// LS Electric XG5000 project: LoadWizardAreopag
// PLC LSPLC
// module base 0 slot 0: FEnet:XGL-EFMT(B) (Fast Ethernet Module, Electrical Master)
// module base 0 slot 1: Input Module:XGI-D24A/B (DC 24V Input, 32 Contacts)
// module base 0 slot 2: Output Module:XGQ-TR4A/B (Transistor Output, 32 Contacts (0.1A, Sink Output/Source Output))
// module base 0 slot 3: 64points reservation:XG-IN64

PROGRAM Main (task: Scan Program)

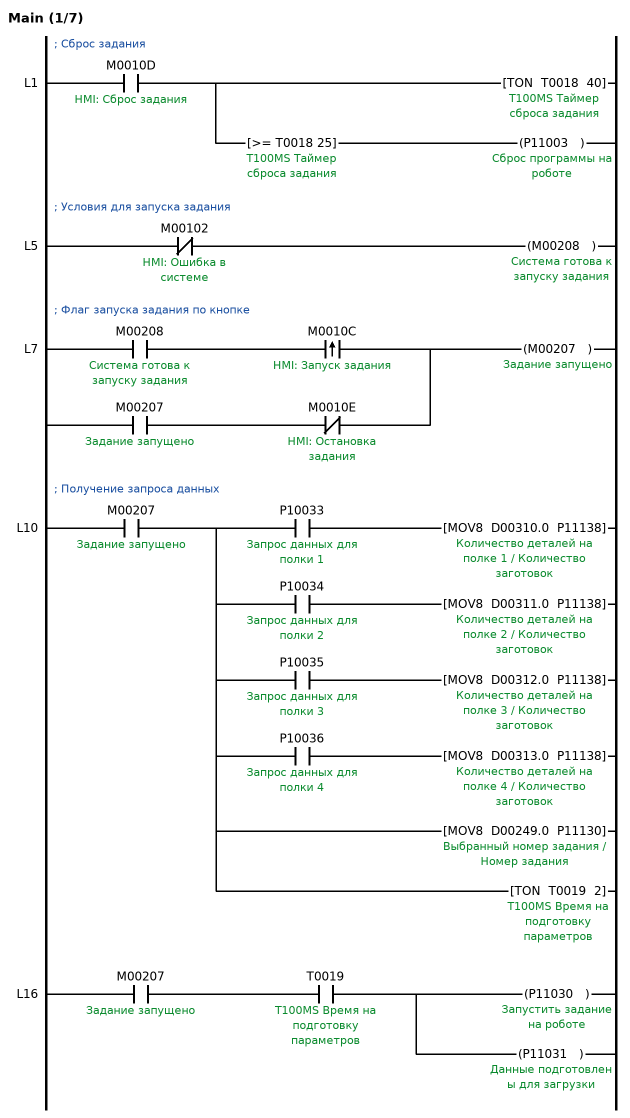
// Сброс задания
; L1
LOAD      M0010D	// HMI: Сброс задания
TON       T0018 40	// T100MS Таймер сброса задания
AND>=     T0018 25	// T100MS Таймер сброса задания
OUT       P11003	// Сброс программы на роботе
// Условия для запуска задания
; L5
LOAD NOT  M00102	// HMI: Ошибка в системе
OUT       M00208	// Система готова к запуску задания
// Флаг запуска задания по кнопке
; L7
LOAD      M00208	// Система готова к запуску задания
ANDP      M0010C	// HMI: Запуск задания
LOAD      M00207	// Задание запущено
AND NOT   M0010E	// HMI: Остановка задания
OR LOAD
OUT       M00207	// Задание запущено
// Получение запроса данных
; L10
LOAD      M00207	// Задание запущено
MPUSH
AND       P10033	// Запрос данных для полки 1
MOV8      D00310.0 P11138	// Количество деталей на полке 1 / Количество заготовок
MLOAD
AND       P10034	// Запрос данных для полки 2
MOV8      D00311.0 P11138	// Количество деталей на полке 2 / Количество заготовок
MLOAD
AND       P10035	// Запрос данных для полки 3
MOV8      D00312.0 P11138	// Количество деталей на полке 3 / Количество заготовок
MLOAD
AND       P10036	// Запрос данных для полки 4
MOV8      D00313.0 P11138	// Количество деталей на полке 4 / Количество заготовок
MPOP
MOV8      D00249.0 P11130	// Выбранный номер задания / Номер задания
TON       T0019 2	// T100MS Время на подготовку параметров
; L16
LOAD      M00207	// Задание запущено
AND       T0019	// T100MS Время на подготовку параметров
OUT       P11030	// Запустить задание на роботе
OUT       P11031	// Данные подготовлены для загрузки

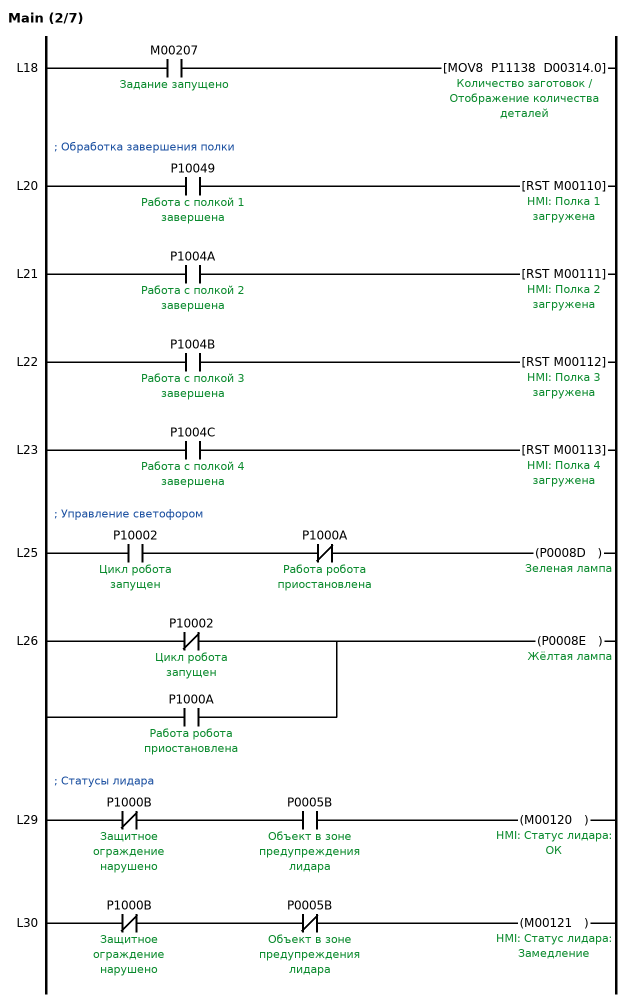
; L18
LOAD      M00207	// Задание запущено
MOV8      P11138 D00314.0	// Количество заготовок / Отображение количества деталей
// Обработка завершения полки
; L20
LOAD      P10049	// Работа с полкой 1 завершена
RST       M00110	// HMI: Полка 1 загружена
; L21
LOAD      P1004A	// Работа с полкой 2 завершена
RST       M00111	// HMI: Полка 2 загружена
; L22
LOAD      P1004B	// Работа с полкой 3 завершена
RST       M00112	// HMI: Полка 3 загружена
; L23
LOAD      P1004C	// Работа с полкой 4 завершена
RST       M00113	// HMI: Полка 4 загружена
// Управление светофором
; L25
LOAD      P10002	// Цикл робота запущен
AND NOT   P1000A	// Работа робота приостановлена
OUT       P0008D	// Зеленая лампа
; L26
LOAD NOT  P10002	// Цикл робота запущен
OR        P1000A	// Работа робота приостановлена
OUT       P0008E	// Жёлтая лампа
// Статусы лидара
; L29
LOAD NOT  P1000B	// Защитное ограждение нарушено
AND       P0005B	// Объект в зоне предупреждения лидара
OUT       M00120	// HMI: Статус лидара: ОК
; L30
LOAD NOT  P1000B	// Защитное ограждение нарушено
AND NOT   P0005B	// Объект в зоне предупреждения лидара
OUT       M00121	// HMI: Статус лидара: Замедление

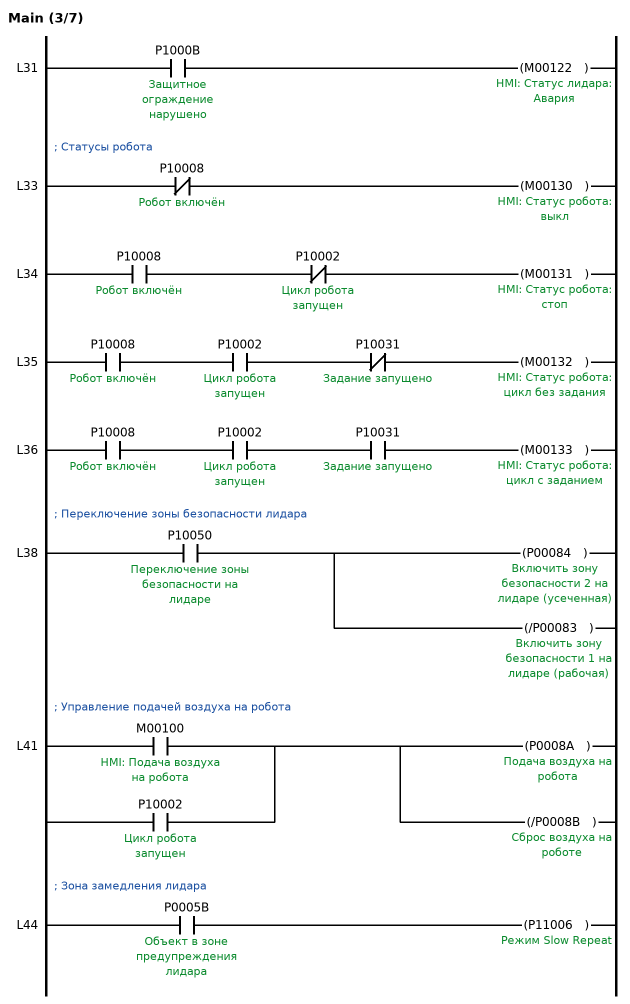
; L31
LOAD      P1000B	// Защитное ограждение нарушено
OUT       M00122	// HMI: Статус лидара: Авария
// Статусы робота
; L33
LOAD NOT  P10008	// Робот включён
OUT       M00130	// HMI: Статус робота: выкл
; L34
LOAD      P10008	// Робот включён
AND NOT   P10002	// Цикл робота запущен
OUT       M00131	// HMI: Статус робота: стоп
; L35
LOAD      P10008	// Робот включён
AND       P10002	// Цикл робота запущен
AND NOT   P10031	// Задание запущено
OUT       M00132	// HMI: Статус робота: цикл без задания
; L36
LOAD      P10008	// Робот включён
AND       P10002	// Цикл робота запущен
AND       P10031	// Задание запущено
OUT       M00133	// HMI: Статус робота: цикл с заданием
// Переключение зоны безопасности лидара 
; L38
LOAD      P10050	// Переключение зоны безопасности на лидаре
OUT       P00084	// Включить зону безопасности 2 на лидаре (усеченная)
OUT NOT   P00083	// Включить зону безопасности 1 на лидаре (рабочая)
// Управление подачей воздуха на робота
; L41
LOAD      M00100	// HMI: Подача воздуха на робота
OR        P10002	// Цикл робота запущен
OUT       P0008A	// Подача воздуха на робота
OUT NOT   P0008B	// Сброс воздуха на роботе
// Зона замедления лидара
; L44
LOAD      P0005B	// Объект в зоне предупреждения лидара
OUT       P11006	// Режим Slow Repeat

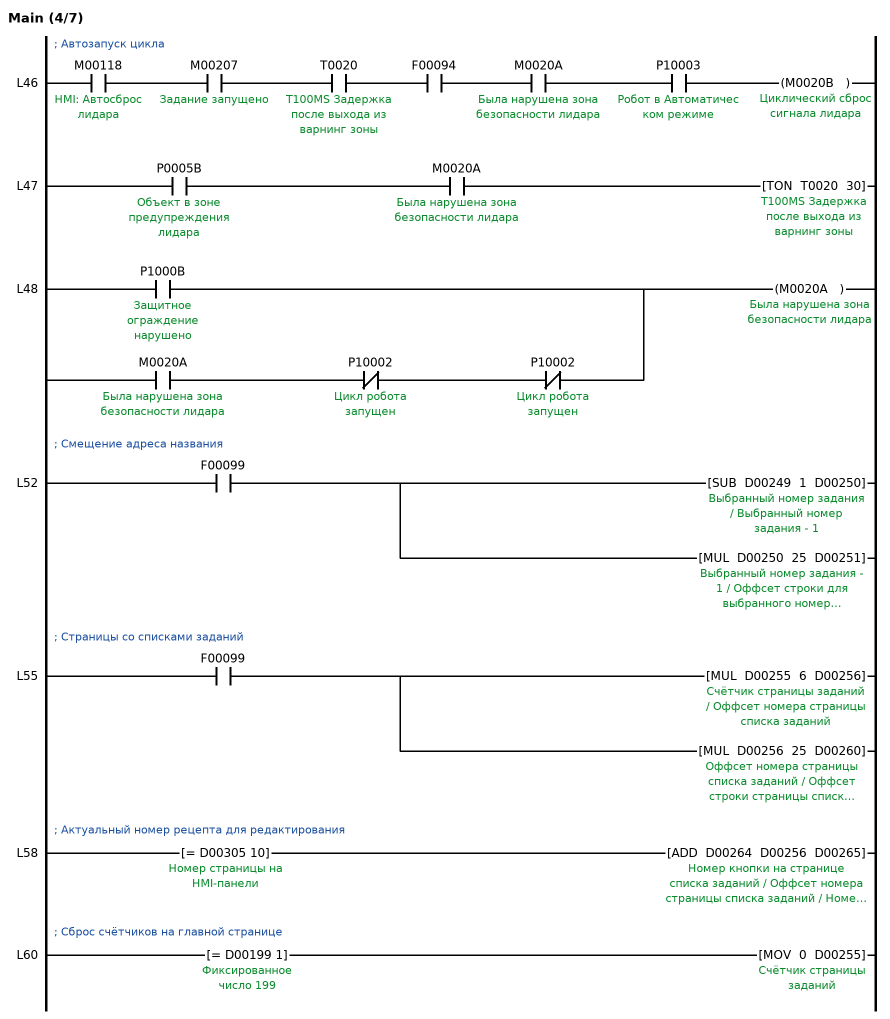
// Автозапуск цикла
; L46
LOAD      M00118	// HMI: Автосброс лидара
AND       M00207	// Задание запущено
AND       T0020	// T100MS Задержка после выхода из варнинг зоны
AND       F00094
AND       M0020A	// Была нарушена зона безопасности лидара
AND       P10003	// Робот в Автоматическом режиме
OUT       M0020B	// Циклический сброс сигнала лидара
; L47
LOAD      P0005B	// Объект в зоне предупреждения лидара
AND       M0020A	// Была нарушена зона безопасности лидара
TON       T0020 30	// T100MS Задержка после выхода из варнинг зоны
; L48
LOAD      P1000B	// Защитное ограждение нарушено
LOAD      M0020A	// Была нарушена зона безопасности лидара
AND NOT   P10002	// Цикл робота запущен
AND NOT   P10002	// Цикл робота запущен
OR LOAD
OUT       M0020A	// Была нарушена зона безопасности лидара
// Смещение адреса названия
; L52
LOAD      F00099
SUB       D00249 1 D00250	// Выбранный номер задания / Выбранный номер задания - 1
MUL       D00250 25 D00251	// Выбранный номер задания - 1 / Оффсет строки для выбранного номера названия
// Страницы со списками заданий
; L55
LOAD      F00099
MUL       D00255 6 D00256	// Счётчик страницы заданий / Оффсет номера страницы списка заданий
MUL       D00256 25 D00260	// Оффсет номера страницы списка заданий / Оффсет строки страницы списка заданий
// Актуальный номер рецепта для редактирования
; L58
LOAD=     D00305 10	// Номер страницы на HMI-панели
ADD       D00264 D00256 D00265	// Номер кнопки на странице списка заданий / Оффсет номера страницы списка заданий / Номер редактируемого задания
// Сброс счётчиков на главной странице
; L60
LOAD=     D00199 1	// Фиксированное число 199
MOV       0 D00255	// Счётчик страницы заданий

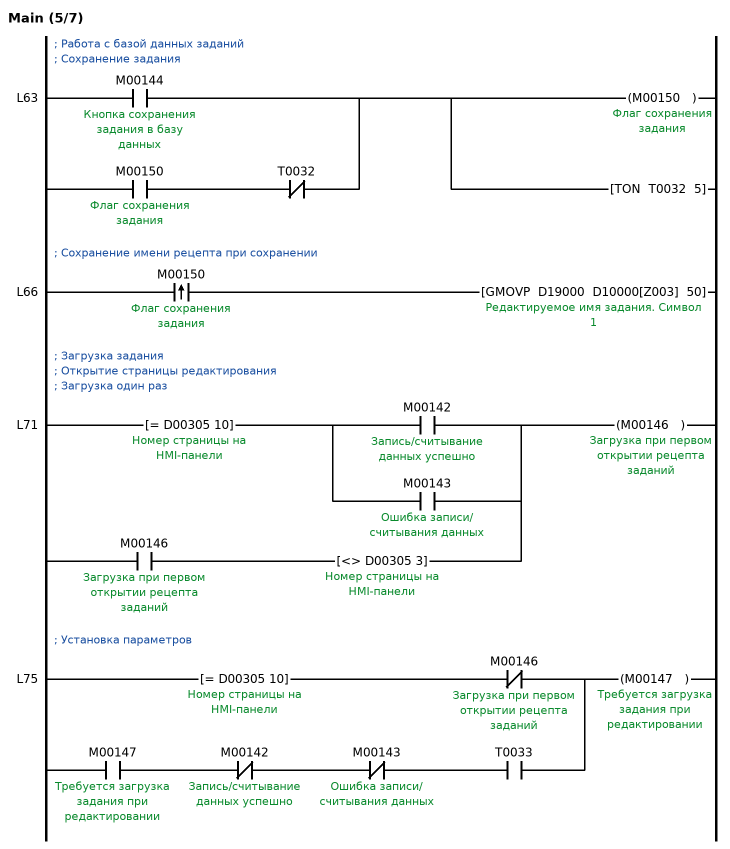
// Работа с базой данных заданий
// Сохранение задания
; L63
LOAD      M00144	// Кнопка сохранения задания в базу данных
LOAD      M00150	// Флаг сохранения задания
AND NOT   T0032
OR LOAD
OUT       M00150	// Флаг сохранения задания
TON       T0032 5
// Сохранение имени рецепта при сохранении
; L66
LOADP     M00150	// Флаг сохранения задания
GMOVP     D19000 D10000[Z003] 50	// Редактируемое имя задания. Символ 1
// Загрузка задания
// Открытие страницы редактирования
// Загрузка один раз
; L71
LOAD=     D00305 10	// Номер страницы на HMI-панели
LOAD      M00142	// Запись/считывание данных успешно
OR        M00143	// Ошибка записи/считывания данных
AND LOAD
LOAD      M00146	// Загрузка при первом открытии рецепта заданий
AND<>     D00305 3	// Номер страницы на HMI-панели
OR LOAD
OUT       M00146	// Загрузка при первом открытии рецепта заданий
// Установка параметров
; L75
LOAD=     D00305 10	// Номер страницы на HMI-панели
AND NOT   M00146	// Загрузка при первом открытии рецепта заданий
LOAD      M00147	// Требуется загрузка задания при редактировании
AND NOT   M00142	// Запись/считывание данных успешно
AND NOT   M00143	// Ошибка записи/считывания данных
AND       T0033
OR LOAD
OUT       M00147	// Требуется загрузка задания при редактировании

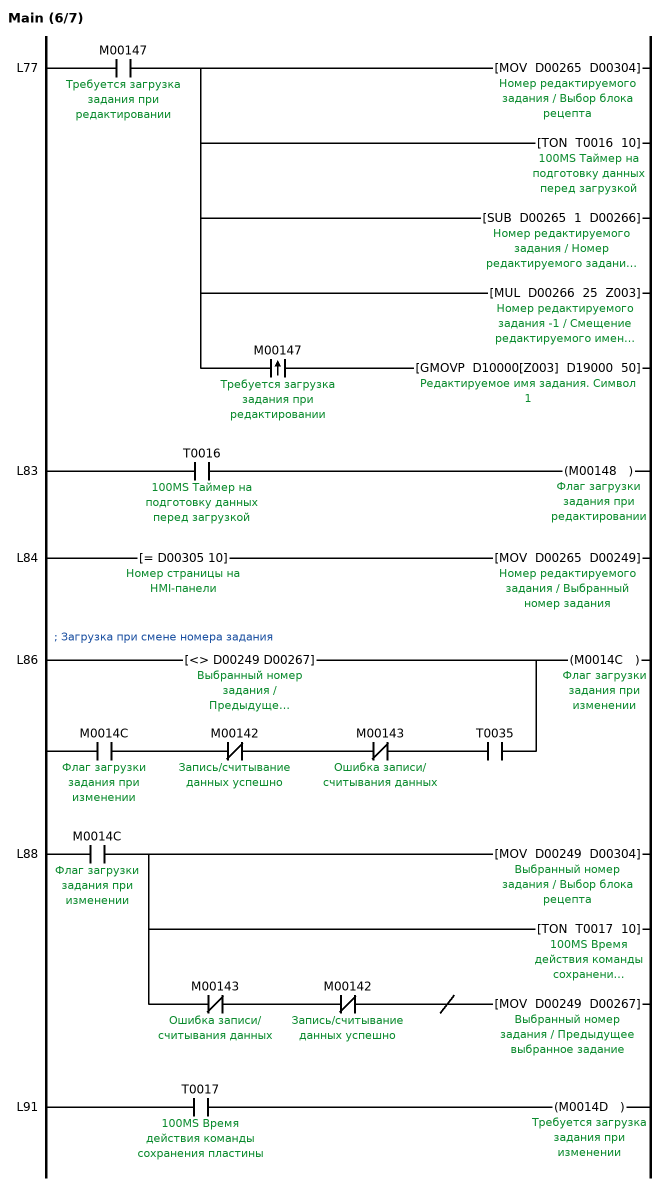
; L77
LOAD      M00147	// Требуется загрузка задания при редактировании
MOV       D00265 D00304	// Номер редактируемого задания / Выбор блока рецепта
TON       T0016 10	// 100MS Таймер на подготовку данных перед загрузкой
SUB       D00265 1 D00266	// Номер редактируемого задания / Номер редактируемого задания -1
MUL       D00266 25 Z003	// Номер редактируемого задания -1 / Смещение редактируемого имени задания
ANDP      M00147	// Требуется загрузка задания при редактировании
GMOVP     D10000[Z003] D19000 50	// Редактируемое имя задания. Символ 1
; L83
LOAD      T0016	// 100MS Таймер на подготовку данных перед загрузкой
OUT       M00148	// Флаг загрузки задания при редактировании
; L84
LOAD=     D00305 10	// Номер страницы на HMI-панели
MOV       D00265 D00249	// Номер редактируемого задания / Выбранный номер задания
// Загрузка при смене номера задания
; L86
LOAD<>    D00249 D00267	// Выбранный номер задания / Предыдущее выбранное задание
LOAD      M0014C	// Флаг загрузки задания при изменении
AND NOT   M00142	// Запись/считывание данных успешно
AND NOT   M00143	// Ошибка записи/считывания данных
AND       T0035
OR LOAD
OUT       M0014C	// Флаг загрузки задания при изменении
; L88
LOAD      M0014C	// Флаг загрузки задания при изменении
MOV       D00249 D00304	// Выбранный номер задания / Выбор блока рецепта
TON       T0017 10	// 100MS Время действия команды сохранения пластины
AND NOT   M00143	// Ошибка записи/считывания данных
AND NOT   M00142	// Запись/считывание данных успешно
NOT
MOV       D00249 D00267	// Выбранный номер задания / Предыдущее выбранное задание
; L91
LOAD      T0017	// 100MS Время действия команды сохранения пластины
OUT       M0014D	// Требуется загрузка задания при изменении

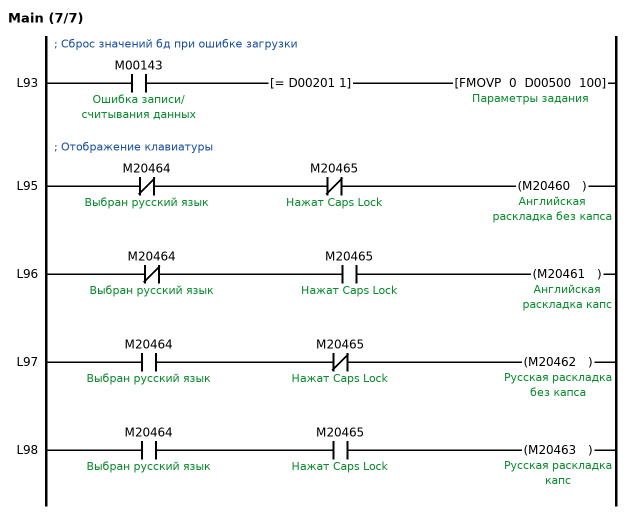
// Сброс значений бд при ошибке загрузки
; L93
LOAD      M00143	// Ошибка записи/считывания данных
AND=      D00201 1
FMOVP     0 D00500 100	// Параметры задания
// Отображение клавиатуры
; L95
LOAD NOT  M20464	// Выбран русский язык
AND NOT   M20465	// Нажат Caps Lock
OUT       M20460	// Английская раскладка без капса
; L96
LOAD NOT  M20464	// Выбран русский язык
AND       M20465	// Нажат Caps Lock
OUT       M20461	// Английская раскладка капс
; L97
LOAD      M20464	// Выбран русский язык
AND NOT   M20465	// Нажат Caps Lock
OUT       M20462	// Русская раскладка без капса
; L98
LOAD      M20464	// Выбран русский язык
AND       M20465	// Нажат Caps Lock
OUT       M20463	// Русская раскладка капс

PROGRAM CNC (task: Scan Program)

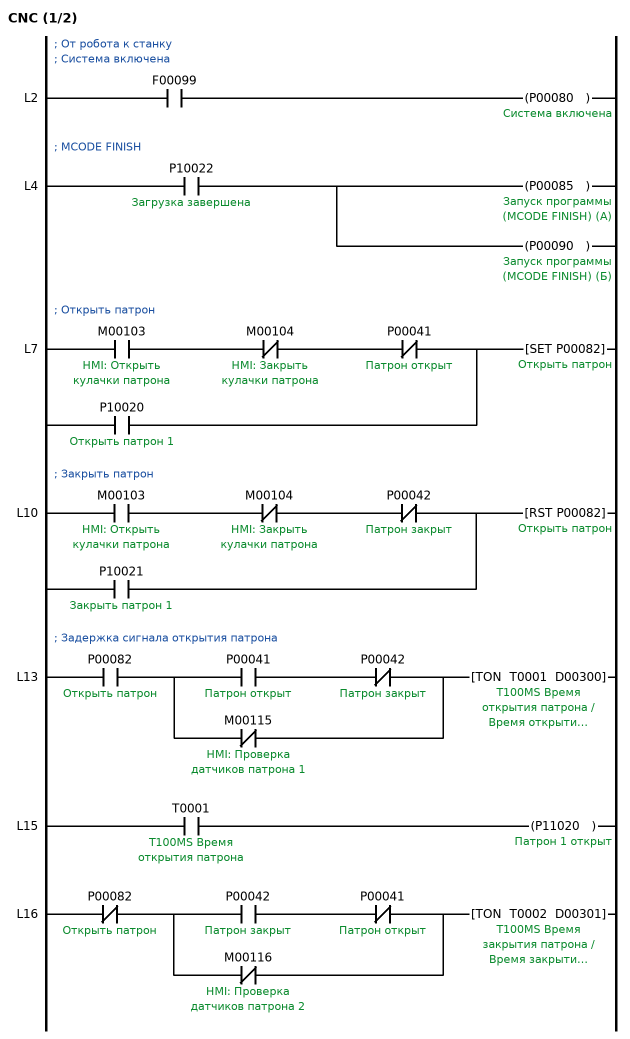
// От робота к станку
// Система включена
; L2
LOAD      F00099
OUT       P00080	// Система включена
// MCODE FINISH
; L4
LOAD      P10022	// Загрузка завершена
OUT       P00085	// Запуск программы (MCODE FINISH) (А)
OUT       P00090	// Запуск программы (MCODE FINISH) (Б)
// Открыть патрон
; L7
LOAD      M00103	// HMI: Открыть кулачки патрона
AND NOT   M00104	// HMI: Закрыть кулачки патрона
AND NOT   P00041	// Патрон открыт
OR        P10020	// Открыть патрон 1
SET       P00082	// Открыть патрон
// Закрыть патрон
; L10
LOAD      M00103	// HMI: Открыть кулачки патрона
AND NOT   M00104	// HMI: Закрыть кулачки патрона
AND NOT   P00042	// Патрон закрыт
OR        P10021	// Закрыть патрон 1
RST       P00082	// Открыть патрон
// Задержка сигнала открытия патрона
; L13
LOAD      P00082	// Открыть патрон
LOAD      P00041	// Патрон открыт
AND NOT   P00042	// Патрон закрыт
OR NOT    M00115	// HMI: Проверка датчиков патрона 1
AND LOAD
TON       T0001 D00300	// T100MS Время открытия патрона / Время открытия патрона (сек)
; L15
LOAD      T0001	// T100MS Время открытия патрона
OUT       P11020	// Патрон 1 открыт
; L16
LOAD NOT  P00082	// Открыть патрон
LOAD      P00042	// Патрон закрыт
AND NOT   P00041	// Патрон открыт
OR NOT    M00116	// HMI: Проверка датчиков патрона 2
AND LOAD
TON       T0002 D00301	// T100MS Время закрытия патрона / Время закрытия патрона (сек)

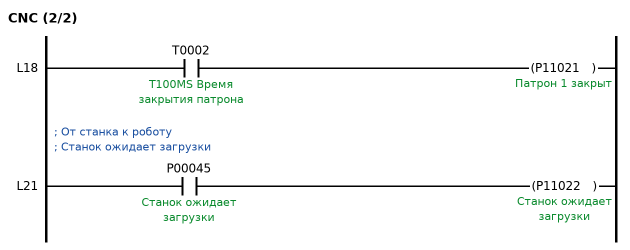
; L18
LOAD      T0002	// T100MS Время закрытия патрона
OUT       P11021	// Патрон 1 закрыт
// От станка к роботу
// Станок ожидает загрузки
; L21
LOAD      P00045	// Станок ожидает загрузки
OUT       P11022	// Станок ожидает загрузки

PROGRAM Error (task: Scan Program)

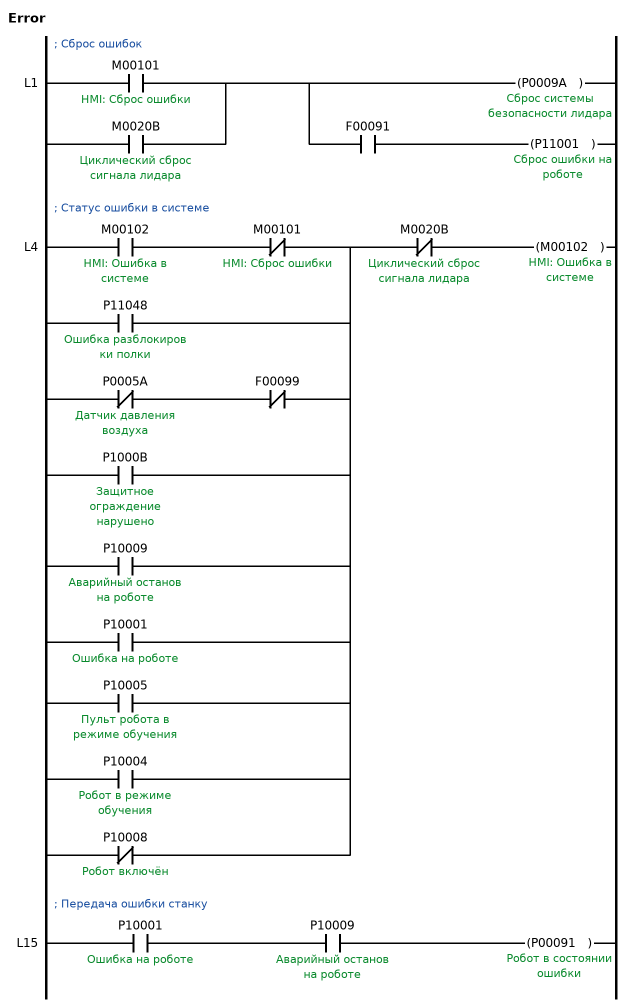
// Сброс ошибок
; L1
LOAD      M00101	// HMI: Сброс ошибки
OR        M0020B	// Циклический сброс сигнала лидара
OUT       P0009A	// Сброс системы безопасности лидара
AND       F00091
OUT       P11001	// Сброс ошибки на роботе
// Статус ошибки в системе
; L4
LOAD      M00102	// HMI: Ошибка в системе
AND NOT   M00101	// HMI: Сброс ошибки
OR        P11048	// Ошибка разблокировки полки
LOAD NOT  P0005A	// Датчик давления воздуха
AND NOT   F00099
OR LOAD
OR        P1000B	// Защитное ограждение нарушено
OR        P10009	// Аварийный останов на роботе
OR        P10001	// Ошибка на роботе
OR        P10005	// Пульт робота в режиме обучения
OR        P10004	// Робот в режиме обучения
OR NOT    P10008	// Робот включён
AND NOT   M0020B	// Циклический сброс сигнала лидара
OUT       M00102	// HMI: Ошибка в системе
// Передача ошибки станку
; L15
LOAD      P10001	// Ошибка на роботе
AND       P10009	// Аварийный останов на роботе
OUT       P00091	// Робот в состоянии ошибки

PROGRAM Stocker (task: Scan Program)

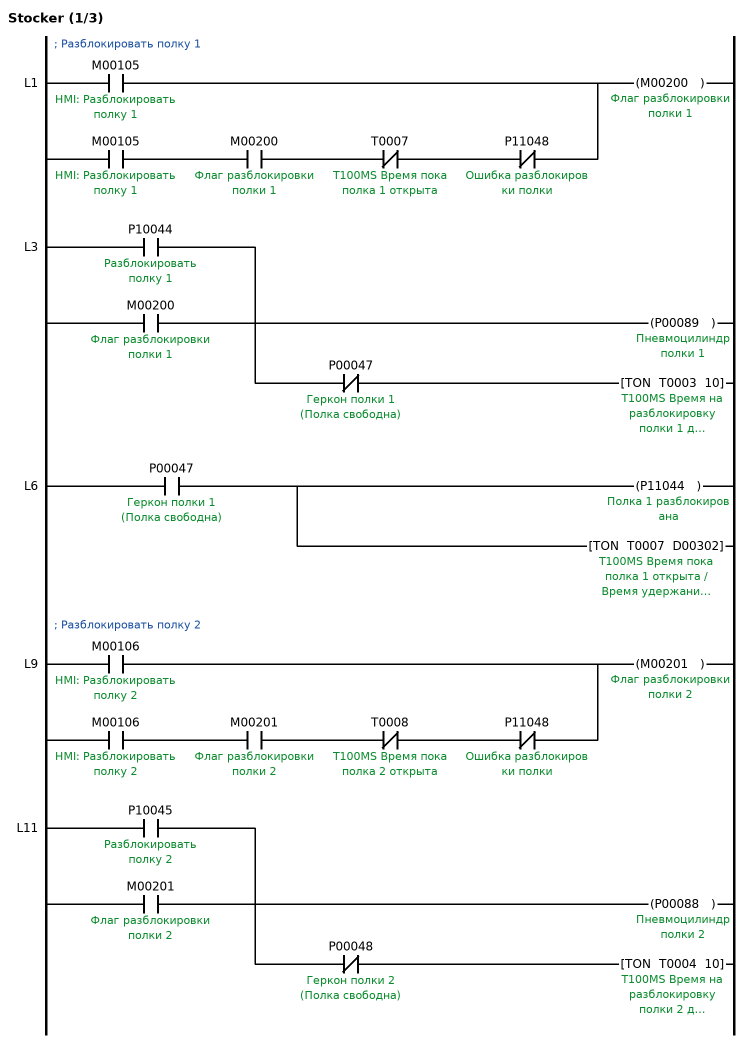
// Разблокировать полку 1
; L1
LOAD      M00105	// HMI: Разблокировать полку 1
LOAD      M00105	// HMI: Разблокировать полку 1
AND       M00200	// Флаг разблокировки полки 1
AND NOT   T0007	// T100MS Время пока полка 1 открыта
AND NOT   P11048	// Ошибка разблокировки полки
OR LOAD
OUT       M00200	// Флаг разблокировки полки 1
; L3
LOAD      P10044	// Разблокировать полку 1
OR        M00200	// Флаг разблокировки полки 1
OUT       P00089	// Пневмоцилиндр полки 1
AND NOT   P00047	// Геркон полки 1 (Полка свободна)
TON       T0003 10	// T100MS Время на разблокировку полки 1 до появления ошибки
; L6
LOAD      P00047	// Геркон полки 1 (Полка свободна)
OUT       P11044	// Полка 1 разблокирована
TON       T0007 D00302	// T100MS Время пока полка 1 открыта / Время удержания полки открытой (сек)
// Разблокировать полку 2
; L9
LOAD      M00106	// HMI: Разблокировать полку 2
LOAD      M00106	// HMI: Разблокировать полку 2
AND       M00201	// Флаг разблокировки полки 2
AND NOT   T0008	// T100MS Время пока полка 2 открыта
AND NOT   P11048	// Ошибка разблокировки полки
OR LOAD
OUT       M00201	// Флаг разблокировки полки 2
; L11
LOAD      P10045	// Разблокировать полку 2
OR        M00201	// Флаг разблокировки полки 2
OUT       P00088	// Пневмоцилиндр полки 2
AND NOT   P00048	// Геркон полки 2 (Полка свободна)
TON       T0004 10	// T100MS Время на разблокировку полки 2 до появления ошибки

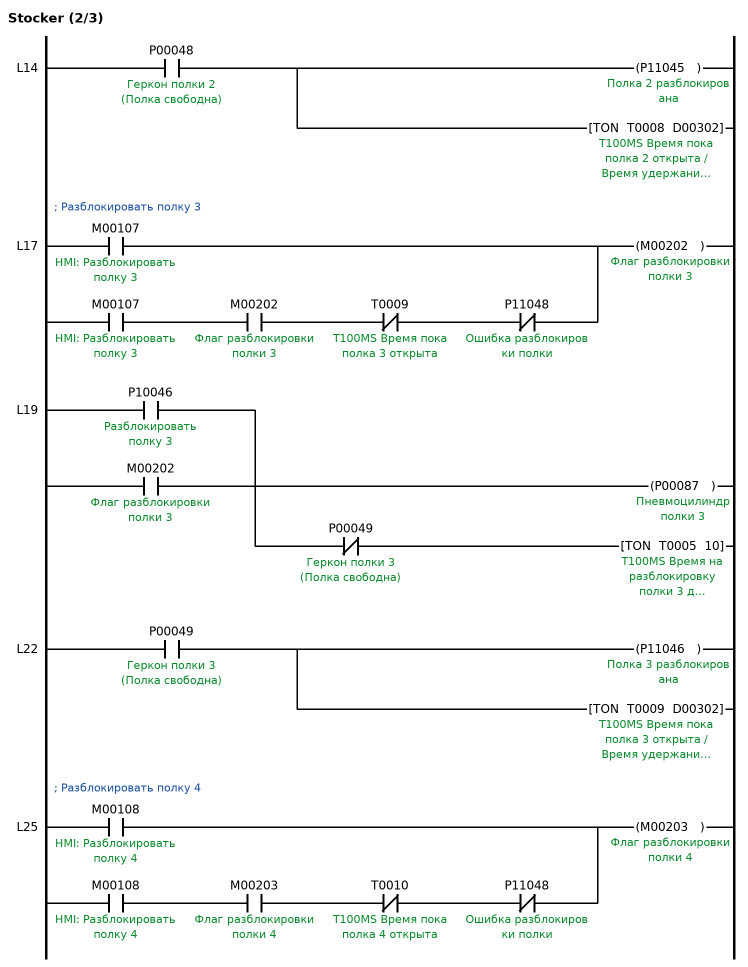
; L14
LOAD      P00048	// Геркон полки 2 (Полка свободна)
OUT       P11045	// Полка 2 разблокирована
TON       T0008 D00302	// T100MS Время пока полка 2 открыта / Время удержания полки открытой (сек)
// Разблокировать полку 3
; L17
LOAD      M00107	// HMI: Разблокировать полку 3
LOAD      M00107	// HMI: Разблокировать полку 3
AND       M00202	// Флаг разблокировки полки 3
AND NOT   T0009	// T100MS Время пока полка 3 открыта
AND NOT   P11048	// Ошибка разблокировки полки
OR LOAD
OUT       M00202	// Флаг разблокировки полки 3
; L19
LOAD      P10046	// Разблокировать полку 3
OR        M00202	// Флаг разблокировки полки 3
OUT       P00087	// Пневмоцилиндр полки 3
AND NOT   P00049	// Геркон полки 3 (Полка свободна)
TON       T0005 10	// T100MS Время на разблокировку полки 3 до появления ошибки
; L22
LOAD      P00049	// Геркон полки 3 (Полка свободна)
OUT       P11046	// Полка 3 разблокирована
TON       T0009 D00302	// T100MS Время пока полка 3 открыта / Время удержания полки открытой (сек)
// Разблокировать полку 4
; L25
LOAD      M00108	// HMI: Разблокировать полку 4
LOAD      M00108	// HMI: Разблокировать полку 4
AND       M00203	// Флаг разблокировки полки 4
AND NOT   T0010	// T100MS Время пока полка 4 открыта
AND NOT   P11048	// Ошибка разблокировки полки
OR LOAD
OUT       M00203	// Флаг разблокировки полки 4

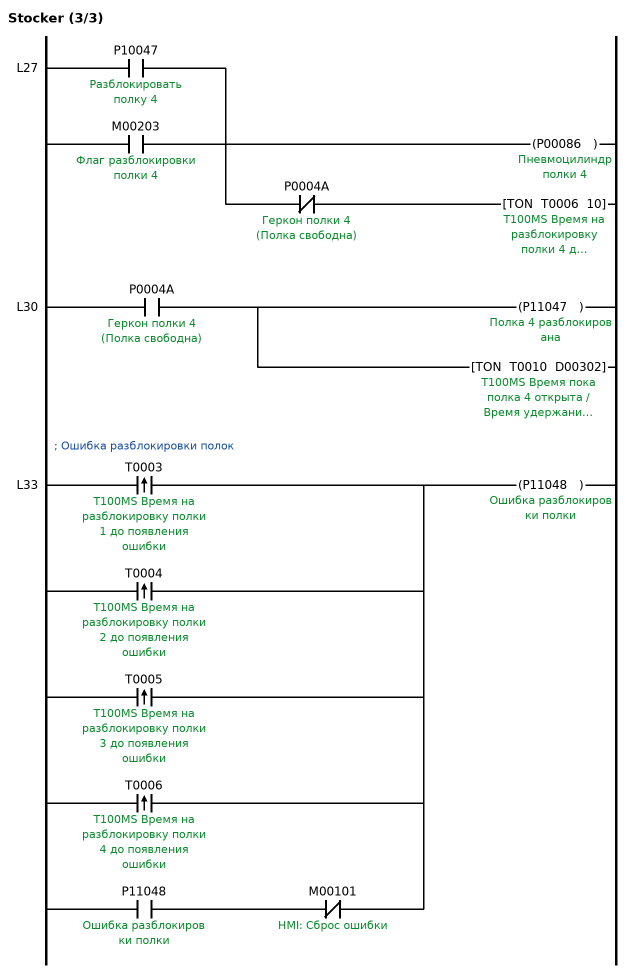
; L27
LOAD      P10047	// Разблокировать полку 4
OR        M00203	// Флаг разблокировки полки 4
OUT       P00086	// Пневмоцилиндр полки 4
AND NOT   P0004A	// Геркон полки 4 (Полка свободна)
TON       T0006 10	// T100MS Время на разблокировку полки 4 до появления ошибки
; L30
LOAD      P0004A	// Геркон полки 4 (Полка свободна)
OUT       P11047	// Полка 4 разблокирована
TON       T0010 D00302	// T100MS Время пока полка 4 открыта / Время удержания полки открытой (сек)
// Ошибка разблокировки полок
; L33
LOADP     T0003	// T100MS Время на разблокировку полки 1 до появления ошибки
ORP       T0004	// T100MS Время на разблокировку полки 2 до появления ошибки
ORP       T0005	// T100MS Время на разблокировку полки 3 до появления ошибки
ORP       T0006	// T100MS Время на разблокировку полки 4 до появления ошибки
LOAD      P11048	// Ошибка разблокировки полки
AND NOT   M00101	// HMI: Сброс ошибки
OR LOAD
OUT       P11048	// Ошибка разблокировки полки

PROGRAM Database (task: Scan Program)

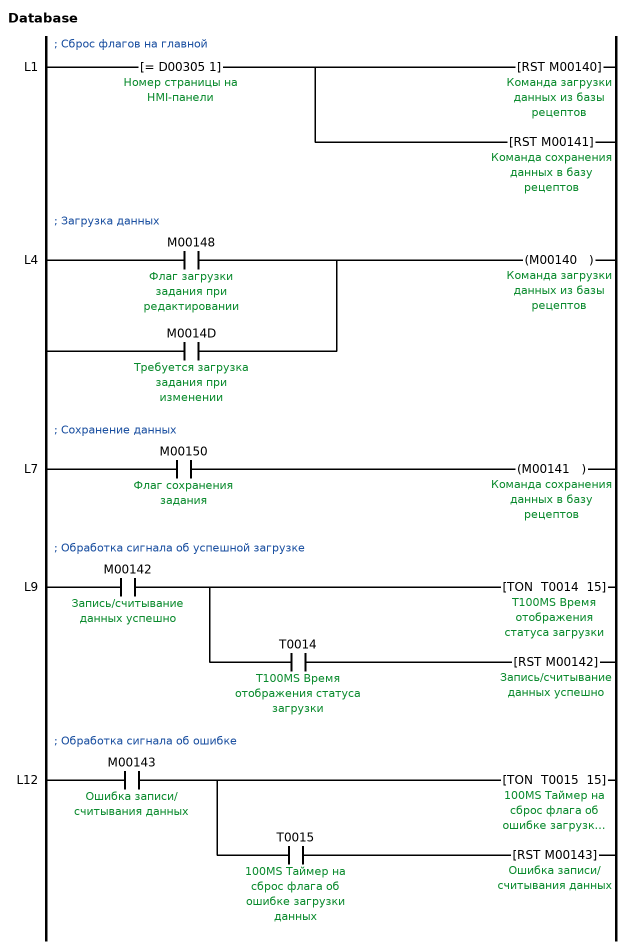
// Сброс флагов на главной
; L1
LOAD=     D00305 1	// Номер страницы на HMI-панели
RST       M00140	// Команда загрузки данных из базы рецептов
RST       M00141	// Команда сохранения данных в базу рецептов
// Загрузка данных
; L4
LOAD      M00148	// Флаг загрузки задания при редактировании
OR        M0014D	// Требуется загрузка задания при изменении
OUT       M00140	// Команда загрузки данных из базы рецептов
// Сохранение данных
; L7
LOAD      M00150	// Флаг сохранения задания
OUT       M00141	// Команда сохранения данных в базу рецептов
// Обработка сигнала об успешной загрузке
; L9
LOAD      M00142	// Запись/считывание данных успешно
TON       T0014 15	// T100MS Время отображения статуса загрузки
AND       T0014	// T100MS Время отображения статуса загрузки
RST       M00142	// Запись/считывание данных успешно
// Обработка сигнала об ошибке
; L12
LOAD      M00143	// Ошибка записи/считывания данных
TON       T0015 15	// 100MS Таймер на сброс флага об ошибке загрузки данных
AND       T0015	// 100MS Таймер на сброс флага об ошибке загрузки данных
RST       M00143	// Ошибка записи/считывания данных

PROGRAM Initialization (task: Scan Program)

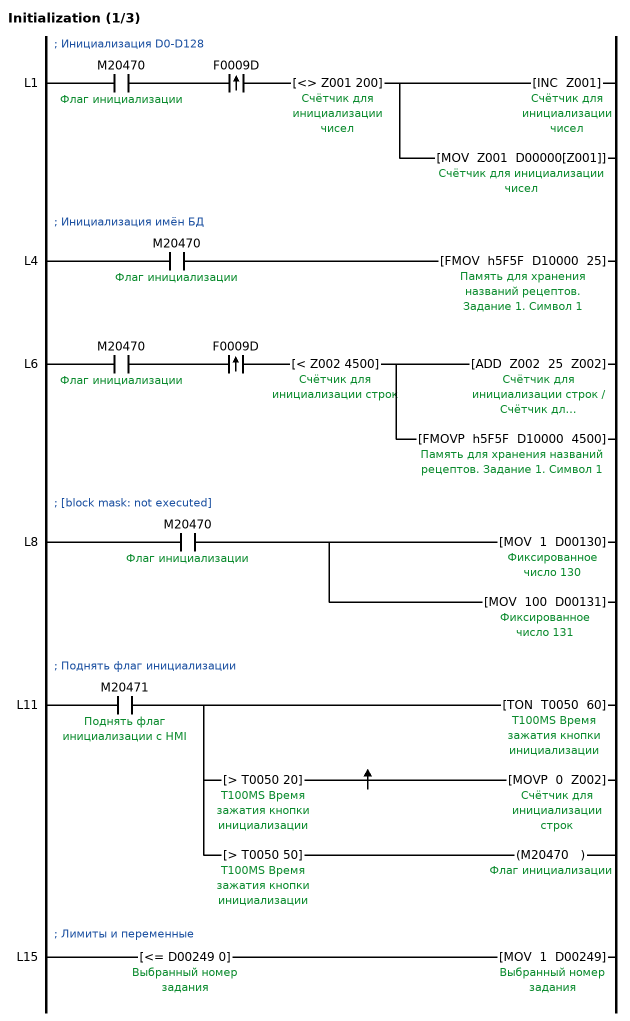
// Инициализация D0-D128
; L1
LOAD      M20470	// Флаг инициализации
ANDP      F0009D
AND<>     Z001 200	// Счётчик для инициализации чисел
INC       Z001	// Счётчик для инициализации чисел
MOV       Z001 D00000[Z001]	// Счётчик для инициализации чисел
// Инициализация имён БД
; L4
LOAD      M20470	// Флаг инициализации
FMOV      h5F5F D10000 25	// Память для хранения названий рецептов. Задание 1. Символ 1
; L6
LOAD      M20470	// Флаг инициализации
ANDP      F0009D
AND<      Z002 4500	// Счётчик для инициализации строк
ADD       Z002 25 Z002	// Счётчик для инициализации строк / Счётчик для инициализации строк
FMOVP     h5F5F D10000 4500	// Память для хранения названий рецептов. Задание 1. Символ 1
; L8 (block mask: not executed)
LOAD      M20470	// Флаг инициализации
MOV       1 D00130	// Фиксированное число 130
MOV       100 D00131	// Фиксированное число 131
// Поднять флаг инициализации
; L11
LOAD      M20471	// Поднять флаг инициализации с HMI
TON       T0050 60	// T100MS Время зажатия кнопки инициализации
MPUSH
AND>      T0050 20	// T100MS Время зажатия кнопки инициализации
R_EDGE
MOVP      0 Z002	// Счётчик для инициализации строк
MPOP
AND>      T0050 50	// T100MS Время зажатия кнопки инициализации
OUT       M20470	// Флаг инициализации
// Лимиты и переменные
; L15
LOAD<=    D00249 0	// Выбранный номер задания
MOV       1 D00249	// Выбранный номер задания

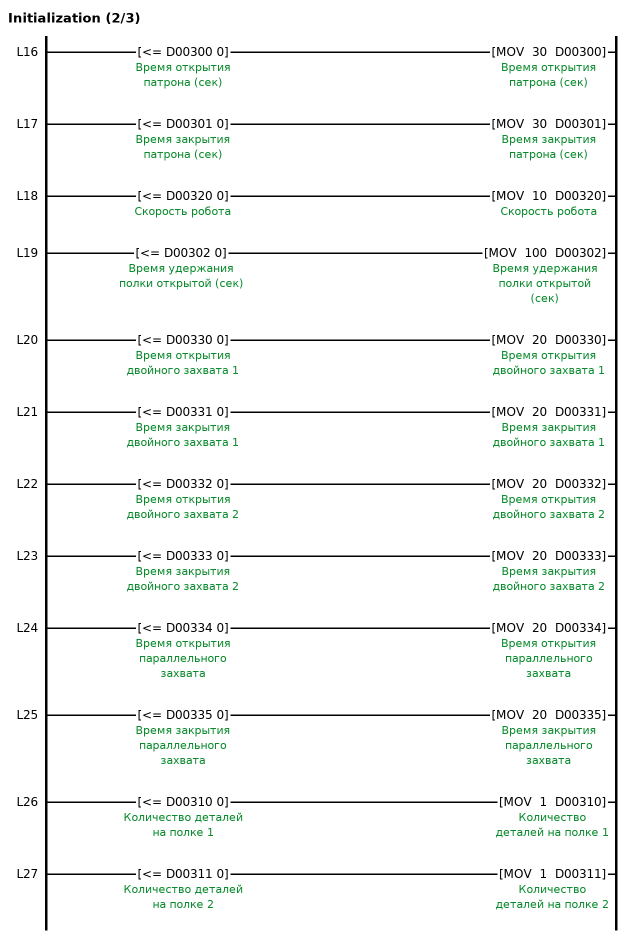
; L16
LOAD<=    D00300 0	// Время открытия патрона (сек)
MOV       30 D00300	// Время открытия патрона (сек)
; L17
LOAD<=    D00301 0	// Время закрытия патрона (сек)
MOV       30 D00301	// Время закрытия патрона (сек)
; L18
LOAD<=    D00320 0	// Скорость робота
MOV       10 D00320	// Скорость робота
; L19
LOAD<=    D00302 0	// Время удержания полки открытой (сек)
MOV       100 D00302	// Время удержания полки открытой (сек)
; L20
LOAD<=    D00330 0	// Время открытия двойного захвата 1
MOV       20 D00330	// Время открытия двойного захвата 1
; L21
LOAD<=    D00331 0	// Время закрытия двойного захвата 1
MOV       20 D00331	// Время закрытия двойного захвата 1
; L22
LOAD<=    D00332 0	// Время открытия двойного захвата 2
MOV       20 D00332	// Время открытия двойного захвата 2
; L23
LOAD<=    D00333 0	// Время закрытия двойного захвата 2
MOV       20 D00333	// Время закрытия двойного захвата 2
; L24
LOAD<=    D00334 0	// Время открытия параллельного захвата
MOV       20 D00334	// Время открытия параллельного захвата
; L25
LOAD<=    D00335 0	// Время закрытия параллельного захвата
MOV       20 D00335	// Время закрытия параллельного захвата
; L26
LOAD<=    D00310 0	// Количество деталей на полке 1
MOV       1 D00310	// Количество деталей на полке 1
; L27
LOAD<=    D00311 0	// Количество деталей на полке 2
MOV       1 D00311	// Количество деталей на полке 2

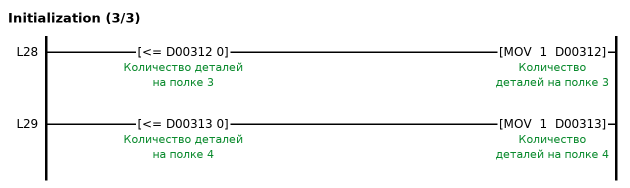
; L28
LOAD<=    D00312 0	// Количество деталей на полке 3
MOV       1 D00312	// Количество деталей на полке 3
; L29
LOAD<=    D00313 0	// Количество деталей на полке 4
MOV       1 D00313	// Количество деталей на полке 4

PROGRAM Robot (task: Scan Program)

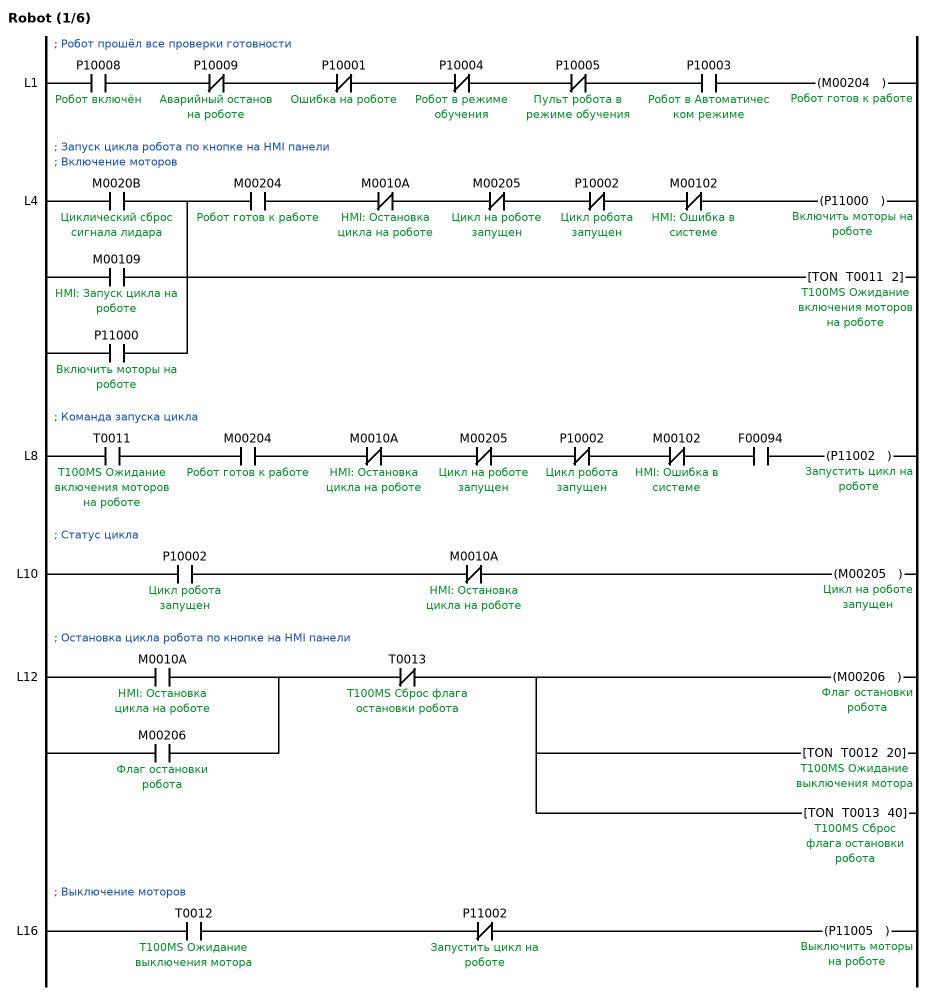
// Робот прошёл все проверки готовности
; L1
LOAD      P10008	// Робот включён
AND NOT   P10009	// Аварийный останов на роботе
AND NOT   P10001	// Ошибка на роботе
AND NOT   P10004	// Робот в режиме обучения
AND NOT   P10005	// Пульт робота в режиме обучения
AND       P10003	// Робот в Автоматическом режиме
OUT       M00204	// Робот готов к работе
// Запуск цикла робота по кнопке на HMI панели
// Включение моторов
; L4
LOAD      M0020B	// Циклический сброс сигнала лидара
OR        M00109	// HMI: Запуск цикла на роботе
OR        P11000	// Включить моторы на роботе
MPUSH
AND       M00204	// Робот готов к работе
AND NOT   M0010A	// HMI: Остановка цикла на роботе
AND NOT   M00205	// Цикл на роботе запущен
AND NOT   P10002	// Цикл робота запущен
AND NOT   M00102	// HMI: Ошибка в системе
OUT       P11000	// Включить моторы на роботе
MPOP
TON       T0011 2	// T100MS Ожидание включения моторов на роботе
// Команда запуска цикла
; L8
LOAD      T0011	// T100MS Ожидание включения моторов на роботе
AND       M00204	// Робот готов к работе
AND NOT   M0010A	// HMI: Остановка цикла на роботе
AND NOT   M00205	// Цикл на роботе запущен
AND NOT   P10002	// Цикл робота запущен
AND NOT   M00102	// HMI: Ошибка в системе
AND       F00094
OUT       P11002	// Запустить цикл на роботе
// Статус цикла
; L10
LOAD      P10002	// Цикл робота запущен
AND NOT   M0010A	// HMI: Остановка цикла на роботе
OUT       M00205	// Цикл на роботе запущен
// Остановка цикла робота по кнопке на HMI панели
; L12
LOAD      M0010A	// HMI: Остановка цикла на роботе
OR        M00206	// Флаг остановки робота
AND NOT   T0013	// T100MS Сброс флага остановки робота
OUT       M00206	// Флаг остановки робота
TON       T0012 20	// T100MS Ожидание выключения мотора
TON       T0013 40	// T100MS Сброс флага остановки робота
// Выключение моторов
; L16
LOAD      T0012	// T100MS Ожидание выключения мотора
AND NOT   P11002	// Запустить цикл на роботе
OUT       P11005	// Выключить моторы на роботе

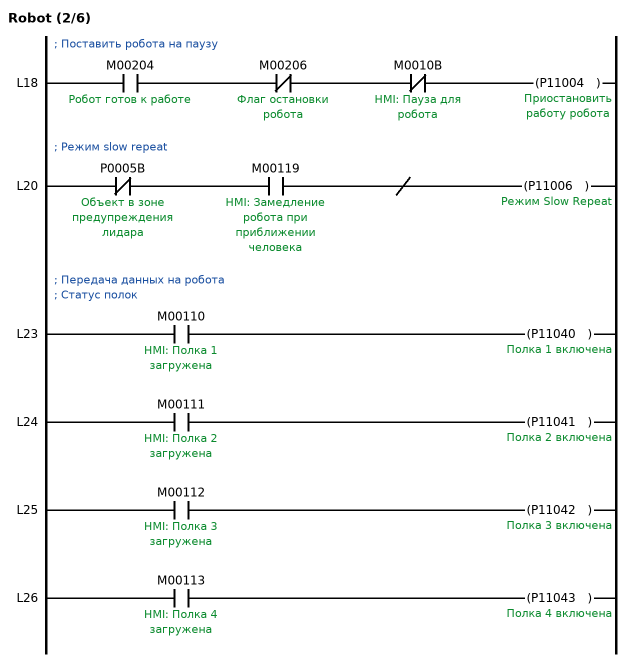
// Поставить робота на паузу
; L18
LOAD      M00204	// Робот готов к работе
AND NOT   M00206	// Флаг остановки робота
AND NOT   M0010B	// HMI: Пауза для робота
OUT       P11004	// Приостановить работу робота
// Режим slow repeat
; L20
LOAD NOT  P0005B	// Объект в зоне предупреждения лидара
AND       M00119	// HMI: Замедление робота при приближении человека
NOT
OUT       P11006	// Режим Slow Repeat
// Передача данных на робота
// Статус полок
; L23
LOAD      M00110	// HMI: Полка 1 загружена
OUT       P11040	// Полка 1 включена
; L24
LOAD      M00111	// HMI: Полка 2 загружена
OUT       P11041	// Полка 2 включена
; L25
LOAD      M00112	// HMI: Полка 3 загружена
OUT       P11042	// Полка 3 включена
; L26
LOAD      M00113	// HMI: Полка 4 загружена
OUT       P11043	// Полка 4 включена

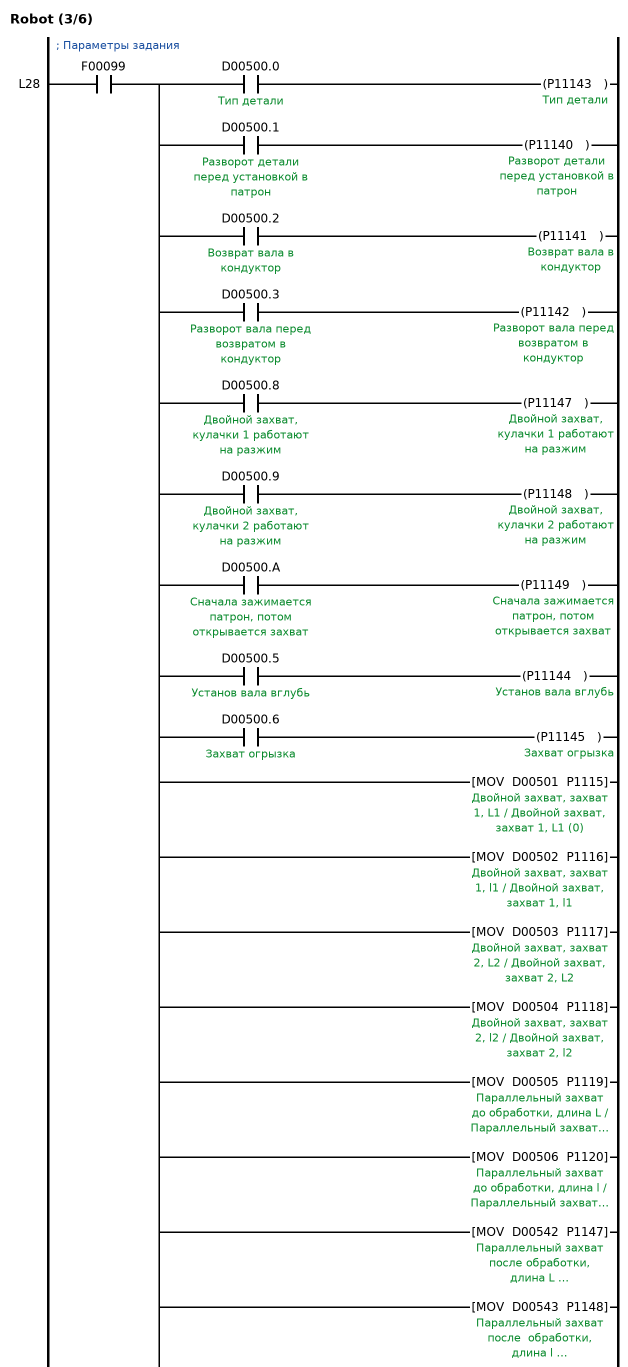

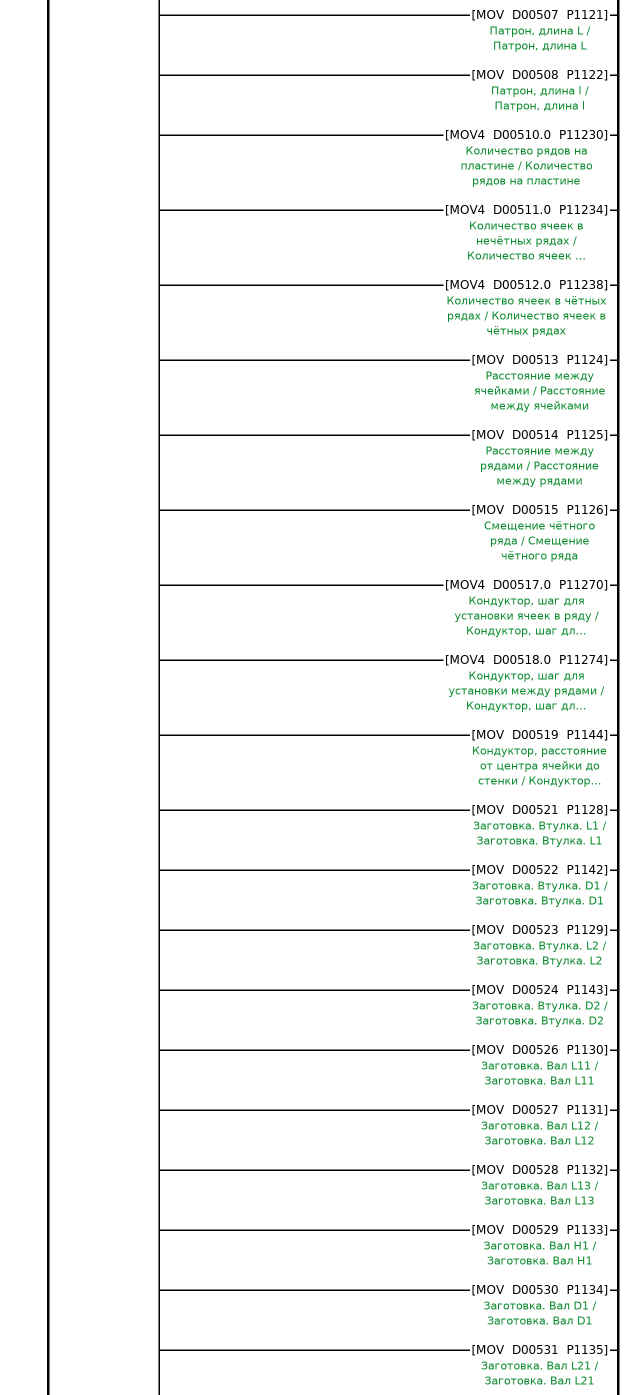

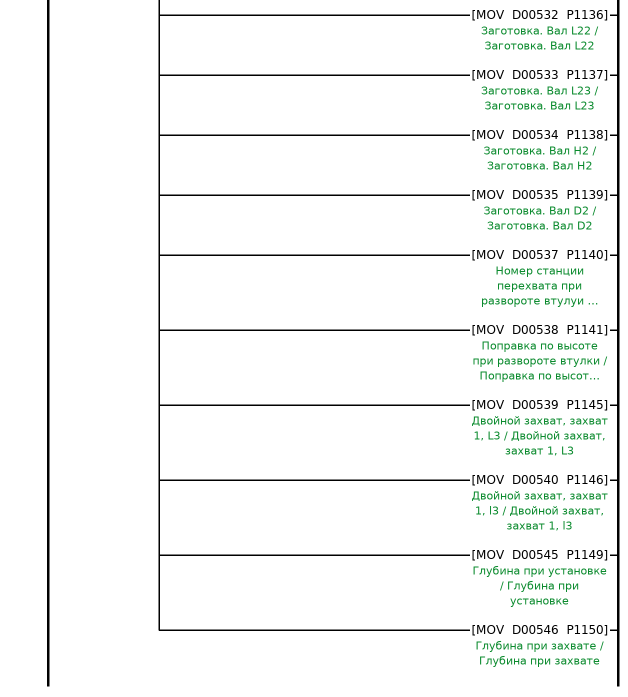
// Параметры задания
; L28
LOAD      F00099
MPUSH
AND       D00500.0	// Тип детали
OUT       P11143	// Тип детали
MLOAD
AND       D00500.1	// Разворот детали перед установкой в патрон
OUT       P11140	// Разворот детали перед установкой в патрон
MLOAD
AND       D00500.2	// Возврат вала в кондуктор
OUT       P11141	// Возврат вала в кондуктор
MLOAD
AND       D00500.3	// Разворот вала перед возвратом в кондуктор
OUT       P11142	// Разворот вала перед возвратом в кондуктор
MLOAD
AND       D00500.8	// Двойной захват, кулачки 1 работают на разжим
OUT       P11147	// Двойной захват, кулачки 1 работают на разжим
MLOAD
AND       D00500.9	// Двойной захват, кулачки 2 работают на разжим
OUT       P11148	// Двойной захват, кулачки 2 работают на разжим
MLOAD
AND       D00500.A	// Сначала зажимается патрон, потом открывается захват
OUT       P11149	// Сначала зажимается патрон, потом открывается захват
MLOAD
AND       D00500.5	// Установ вала вглубь 
OUT       P11144	// Установ вала вглубь
MLOAD
AND       D00500.6	// Захват огрызка
OUT       P11145	// Захват огрызка
MPOP
MOV       D00501 P1115	// Двойной захват, захват 1, L1 / Двойной захват, захват 1, L1 (0)
MOV       D00502 P1116	// Двойной захват, захват 1, l1 / Двойной захват, захват 1, l1
MOV       D00503 P1117	// Двойной захват, захват 2, L2 / Двойной захват, захват 2, L2
MOV       D00504 P1118	// Двойной захват, захват 2, l2 / Двойной захват, захват 2, l2
MOV       D00505 P1119	// Параллельный захват до обработки, длина L / Параллельный захват, до обработки, длина L
MOV       D00506 P1120	// Параллельный захват до обработки, длина l / Параллельный захват, до обработки, длина l
MOV       D00542 P1147	// Параллельный захват после обработки, длина L / Параллельный захват, после обработки, длина L
MOV       D00543 P1148	// Параллельный захват после  обработки, длина l / Параллельный захват, после обработки, длина l
MOV       D00507 P1121	// Патрон, длина L / Патрон, длина L
MOV       D00508 P1122	// Патрон, длина l / Патрон, длина l
MOV4      D00510.0 P11230	// Количество рядов на пластине / Количество рядов на пластине
MOV4      D00511.0 P11234	// Количество ячеек в нечётных рядах / Количество ячеек в нечётных рядах
MOV4      D00512.0 P11238	// Количество ячеек в чётных рядах / Количество ячеек в чётных рядах
MOV       D00513 P1124	// Расстояние между ячейками / Расстояние между ячейками
MOV       D00514 P1125	// Расстояние между рядами / Расстояние между рядами
MOV       D00515 P1126	// Смещение чётного ряда / Смещение чётного ряда
MOV4      D00517.0 P11270	// Кондуктор, шаг для установки ячеек в ряду / Кондуктор, шаг для установки ячеек в ряду
MOV4      D00518.0 P11274	// Кондуктор, шаг для установки между рядами / Кондуктор, шаг для установки между рядами
MOV       D00519 P1144	// Кондуктор, расстояние от центра ячейки до стенки / Кондуктор, расстояние от центра ячейки до стенки
MOV       D00521 P1128	// Заготовка. Втулка. L1 / Заготовка. Втулка. L1
MOV       D00522 P1142	// Заготовка. Втулка. D1 / Заготовка. Втулка. D1
MOV       D00523 P1129	// Заготовка. Втулка. L2 / Заготовка. Втулка. L2
MOV       D00524 P1143	// Заготовка. Втулка. D2 / Заготовка. Втулка. D2
MOV       D00526 P1130	// Заготовка. Вал L11 / Заготовка. Вал L11
MOV       D00527 P1131	// Заготовка. Вал L12 / Заготовка. Вал L12
MOV       D00528 P1132	// Заготовка. Вал L13 / Заготовка. Вал L13
MOV       D00529 P1133	// Заготовка. Вал H1 / Заготовка. Вал H1
MOV       D00530 P1134	// Заготовка. Вал D1 / Заготовка. Вал D1
MOV       D00531 P1135	// Заготовка. Вал L21 / Заготовка. Вал L21
MOV       D00532 P1136	// Заготовка. Вал L22 / Заготовка. Вал L22
MOV       D00533 P1137	// Заготовка. Вал L23 / Заготовка. Вал L23
MOV       D00534 P1138	// Заготовка. Вал H2 / Заготовка. Вал H2
MOV       D00535 P1139	// Заготовка. Вал D2 / Заготовка. Вал D2
MOV       D00537 P1140	// Номер станции перехвата при развороте втулуи / Номер станции перехвата при развороте втулуи
MOV       D00538 P1141	// Поправка по высоте при развороте втулки / Поправка по высоте при развороте втулки
MOV       D00539 P1145	// Двойной захват, захват 1, L3 / Двойной захват, захват 1, L3
MOV       D00540 P1146	// Двойной захват, захват 1, l3 / Двойной захват, захват 1, l3 
MOV       D00545 P1149	// Глубина при установке / Глубина при установке
MOV       D00546 P1150	// Глубина при захвате / Глубина при захвате

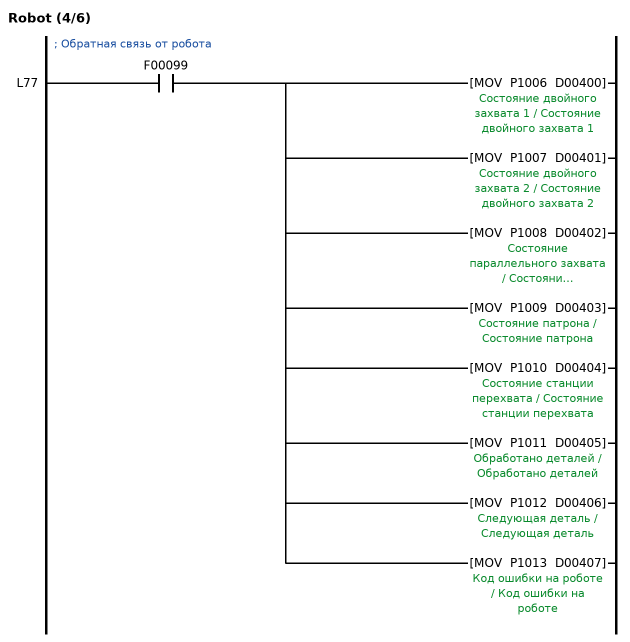
// Обратная связь от робота
; L77
LOAD      F00099
MOV       P1006 D00400	// Состояние двойного захвата 1 / Состояние двойного захвата 1
MOV       P1007 D00401	// Состояние двойного захвата 2 / Состояние двойного захвата 2
MOV       P1008 D00402	// Состояние параллельного захвата / Состояние параллельного захвата
MOV       P1009 D00403	// Состояние патрона / Состояние патрона
MOV       P1010 D00404	// Состояние станции перехвата / Состояние станции перехвата
MOV       P1011 D00405	// Обработано деталей / Обработано деталей
MOV       P1012 D00406	// Следующая деталь / Следующая деталь
MOV       P1013 D00407	// Код ошибки на роботе / Код ошибки на роботе

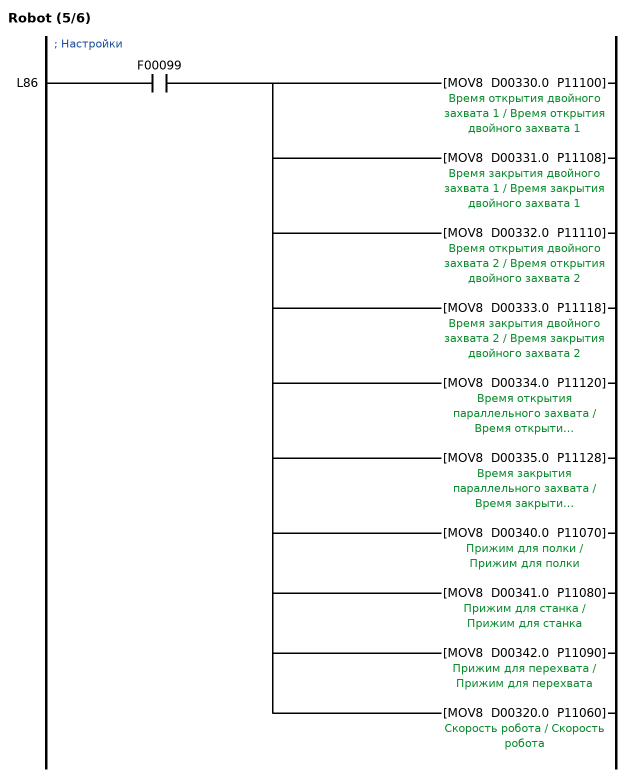
// Настройки
; L86
LOAD      F00099
MOV8      D00330.0 P11100	// Время открытия двойного захвата 1 / Время открытия двойного захвата 1
MOV8      D00331.0 P11108	// Время закрытия двойного захвата 1 / Время закрытия двойного захвата 1
MOV8      D00332.0 P11110	// Время открытия двойного захвата 2 / Время открытия двойного захвата 2
MOV8      D00333.0 P11118	// Время закрытия двойного захвата 2 / Время закрытия двойного захвата 2
MOV8      D00334.0 P11120	// Время открытия параллельного захвата / Время открытия параллельного захвата
MOV8      D00335.0 P11128	// Время закрытия параллельного захвата / Время закрытия параллельного захвата
MOV8      D00340.0 P11070	// Прижим для полки / Прижим для полки
MOV8      D00341.0 P11080	// Прижим для станка / Прижим для станка
MOV8      D00342.0 P11090	// Прижим для перехвата / Прижим для перехвата
MOV8      D00320.0 P11060	// Скорость робота / Скорость робота

